Universal Robots PolyScope program: URControl.urp

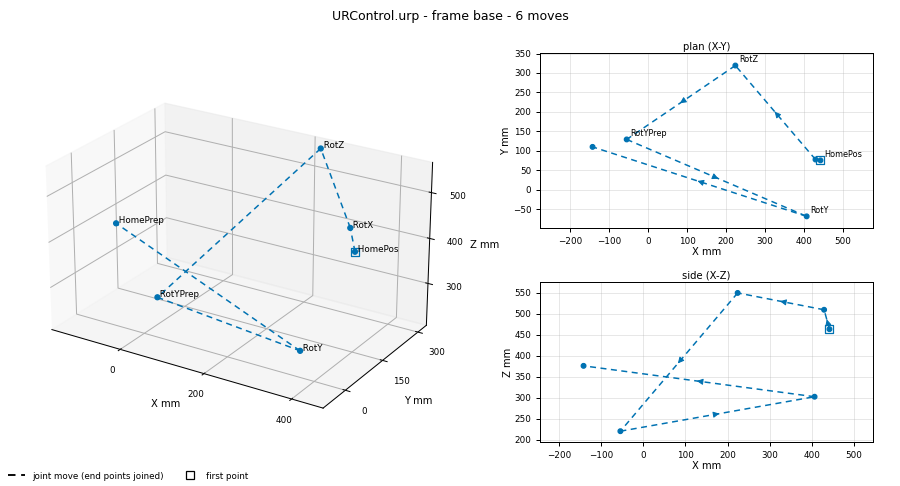
[picture p0: tool path of URControl.urp in frame base, 6 of 6 moves have a stored position in this frame; points joined in program order, loops and branches not executed]
Program Feff (installation=default directory=/programs createdIn=3.13.1.10297 lastSavedIn=3.13.1.10297 robotSerialNumber=2017331984)
Calibrated DH parameters: a=[-0.000081, -0.241371, -0.212703, 0.000038, -0.000013, 0]; d=[0.151828, -12.691906, 15.535277, -2.730958, 0.085254, 0.082431]; alpha=[1.571105, -0.002599, 0.005548, 1.571826, -1.57112, 0]; deltaTheta=[0.000033, 0.135864, -0.061728, -0.07398, -0.000026, 0.000009]
Robot Program (runOnlyOnce=false)
  MoveJ speed 60 deg/s, acceleration 80 deg/s^2 (useActiveTCP=true)
    Waypoint HomePos: TCP in base x=442.243 y=75.844 z=463.387 mm, rx=-1.4199 ry=1.3277 rz=-1.0833 rad; joints [162.258, -17.873, -102.061, -45.987, -70.327, 353.303] deg; flange x=253.996 y=64.588 z=475.869 mm, rx=-1.4199 ry=1.3277 rz=-1.0833 rad
    Wait Sleep waitTime=0.5
  MoveJ speed 60 deg/s, acceleration 80 deg/s^2 (useActiveTCP=true)
    Waypoint RotX: TCP in base x=429.563 y=78.059 z=509.484 mm, rx=-1.3006 ry=1.2159 rz=-1.1824 rad; joints [162.231, -17.866, -102.217, -55.787, -70.325, -3.847] deg; flange x=241.702 y=68.405 z=491.203 mm, rx=-1.3006 ry=1.2159 rz=-1.1824 rad
    Wait Sleep waitTime=0.5
  MoveJ speed 60 deg/s, acceleration 80 deg/s^2 (useActiveTCP=true)
    Waypoint RotZ: TCP in base x=223.995 y=319.159 z=549.501 mm, rx=-1.4656 ry=0.276 rz=0.1369 rad; joints [162.233, -17.763, -98.959, -43.516, -347.026, -3.72] deg; flange x=199.988 y=137.294 z=504.029 mm, rx=-1.4656 ry=0.276 rz=0.1369 rad
    Wait Sleep waitTime=0.5
  MoveJ speed 60 deg/s, acceleration 80 deg/s^2 (useActiveTCP=true)
    Waypoint RotYPrep: TCP in base x=-54.844 y=129.569 z=220.768 mm, rx=-2.1199 ry=-1.7423 rz=0.3338 rad; joints [162.249, -17.792, -101.329, -125.228, -269.875, 353.301] deg; flange x=49.771 y=102.061 z=375.747 mm, rx=-2.1199 ry=-1.7423 rz=0.3338 rad
    Wait Sleep waitTime=0.5
  MoveJ speed 60 deg/s, acceleration 80 deg/s^2 (useActiveTCP=true)
    Waypoint RotY: TCP in base x=406.908 y=-67.762 z=302.743 mm, rx=1.3479 ry=0.9255 rz=0.7539 rad; joints [162.251, -17.794, -96.172, 114.665, -260.322, 353.299] deg; flange x=245.166 y=24.405 z=335.364 mm, rx=1.3479 ry=0.9255 rz=0.7539 rad
    Wait Sleep waitTime=0.5
  MoveJ speed 60 deg/s, acceleration 80 deg/s^2 (useActiveTCP=true)
    Waypoint HomePrep: TCP in base x=-142.371 y=110.45 z=376.158 mm, rx=-1.7123 ry=-1.5389 rz=0.7981 rad; joints [162.253, -24.262, -96.705, -94.469, -260.338, 353.305] deg; flange x=27.419 y=94.553 z=457.632 mm, rx=-1.7123 ry=-1.5389 rz=0.7981 rad
    Wait Sleep waitTime=0.5
